{attribute 'qualified_only'}
TYPE E_PPM_States :
(
    Unknown := 0,
    OUT := 1,
    POWERMETER := 2,
    YAG1 := 3,
    YAG2 := 4
);
END_TYPE

(* stored: Version 1.1.0.1
   DUT E_PPM_States: Id {b72262a0-b857-458c-bac1-465658861dad} *)
